FUNCTION_BLOCK E_N_TABLE (* Generation of a finite train of sperate events *)
  (* Standard: 61499-1 Annex A; Description: Copyright (c) 2017 fortiss GmbH This program and the accompanying materials are made available under the terms of the Eclipse Public License 2.0 which is available at https://www.eclipse.org/legal/epl-2.0/ SPDX-License-Identifier: EPL-2.0 *)
  (* Version 1.0, 2017-09-22, Alois Zoitl, fortiss GmbH, initial API and implementation and/or initial documentation *)
  (* Version 3.0, 2025-04-14, Patrick Aigner, changed package *)
  PACKAGE iec61499::events;
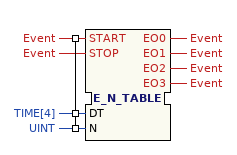
  EVENT_INPUT
    START WITH DT, N;
    STOP;
  END_EVENT
  EVENT_OUTPUT
    EO0;
    EO1;
    EO2;
    EO3;
  END_EVENT
  VAR_INPUT
    DT : ARRAY [0..3] OF TIME;
    N : UINT;
  END_VAR
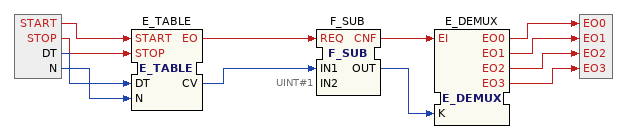
  FBS
    E_TABLE : iec61499::events::E_TABLE;
    E_DEMUX : iec61499::events::E_DEMUX;
    F_SUB : iec61131::arithmetic::F_SUB(IN2 := UINT#1);
  END_FBS
  EVENT_CONNECTIONS
    START TO E_TABLE.START;
    STOP TO E_TABLE.STOP;
    E_TABLE.EO TO F_SUB.REQ;
    F_SUB.CNF TO E_DEMUX.EI;
    E_DEMUX.EO0 TO EO0;
    E_DEMUX.EO1 TO EO1;
    E_DEMUX.EO2 TO EO2;
    E_DEMUX.EO3 TO EO3;
  END_CONNECTIONS
  DATA_CONNECTIONS
    DT TO E_TABLE.DT;
    N TO E_TABLE.N;
    E_TABLE.CV TO F_SUB.IN1;
    F_SUB.OUT TO E_DEMUX.K;
  END_CONNECTIONS
END_FUNCTION_BLOCK
